// Mitsubishi GX Works2 project: plcgroup3_30_1   PLC: FX3G
// plcgroup3

// global labels: Global1
VAR_GLOBAL
  startDay AT X007 : BOOL;  (* מתחיל את היום *)
  ongoingDay AT Y007 : BOOL;  (* נורה שמציינת יום בתהליך *)
  endDay AT X011 : BOOL;  (* מתג סיום יום *)
  hold AT Y007 : BOOL;  (* ממסר החזקה לנורה Y7 *)
  analog_check AT X001 : BOOL;  (* מתג התחלת תהליך בישול *)
  lager AT M2 : BOOL;  (* ערך בינארי שמציין האם נבחר לייצר לאגר *)
  pilzner AT M3 : BOOL;  (* ערך בינארי שמציין האם נבחר לייצר פילסנר *)
  possible_manufacture_lager AT M4 : BOOL;  (* יהיה אחד אם ניתן לייצר לאגר מבחינת מלאי *)
  possible_manufacture_pilzner AT M5 : BOOL;  (* יהיה אחד אם ניתן לייצר פילסנר מבחינת מלאי *)
  cooking_In_process AT Y001 : BOOL;  (* נורה שמציינת שתהליך הבישול מתקיים *)
END_VAR
VAR_GLOBAL CONSTANT
  shmarim_Input_Amount : INT := 1000;  (* קבוע מלאי שמרים שיוזן בתחילת יום *)
  letet_Input_Amount : INT := 400;  (* קבוע מלאי לתת שיוזן בתחילת יום *)
  kashot_input_Amount : INT := 400;  (* קבוע מלאי קשות שיוזן בתחילת יום *)
END_VAR
VAR_GLOBAL
  shmarim_Inventory AT D1130 : INT;  (* רגיסטר שמחזיק בערך מלאי השמרים *)
  letet_Inventory AT D1140 : INT;  (* רגיסטר שמחזיק בערך מלאי הלתת *)
  kashot_Inventory AT D1150 : INT;  (* רגיסטר שמחזיק בערך מלאי הקשות *)
  total_beer_packs AT D1160 : INT;  (* רגיסטר שמחזיק בסך השישיות שיוצרו *)
  analog_Output AT D8282 : INT;  (* אנאלוג אאוטפוט *)
  analog_Input AT D8280 : INT;  (* אנאלוג אינפוט *)
  botteling_1Bottle AT X000 : BOOL;  (* מתג שמבקבק בקבוק אחד *)
  start_Botteling AT X002 : BOOL;  (* מתג שמתחיל בקבוק *)
  finish_Bottleing AT M7 : BOOL;  (* ממסר המציין סיום בקבוק *)
  six_Pack_Ligth AT Y002 : BOOL;  (* נורה שתדלק בזמן הבקבוק *)
END_VAR
VAR_GLOBAL CONSTANT
  constant5 : INT := 5;  (* קבוע 5 *)
END_VAR
VAR_GLOBAL
  cook_TIMER AT TC1 : BOOL;  (* משתנה לזמן הבישול *)
END_VAR
VAR_GLOBAL CONSTANT
  constant_40 : INT := 40;  (* מספר קבוע *)
  constant6 : INT := 6;  (* מספר קבוע *)
  pilzner_letet_6_req : INT := 6;  (* כמות לתת נדרשת לשישיית פילזנר *)
  pilzner_shmarim_6_req : INT := 120;  (* כמות שמרים נדרשת לשישיית פילזנר *)
  pilzner_kshot_6_req : INT := 54;  (* כמות קשות נדרשת לשישיית פילזנר *)
  lager_shmarim_6_req : INT := 150;  (* כמות שמרים נדרשת לשישיית לאגר *)
  lager_letet_6_req : INT := 12;  (* כמות לתת נדרשת לשישיית לאגר *)
  lager_kshot_6_req : INT := 60;  (* כמות קשות נדרשת לשישיית לאגר *)
END_VAR
VAR_GLOBAL
  finish_cooking_timer AT TS1 : BOOL;  (* מציין סיום בישול *)
  stast_tsisa AT X005 : BOOL;  (* מתג הפעלת תסיסה *)
  hivhov_round AT M8 : BOOL;  (* ממסר שיתחיל סבב הבהוב נוסף *)
  bulb3_on AT TC2 : BOOL;  (* הפעלת נורה 3 לצורך הבהוב *)
END_VAR
VAR_GLOBAL CONSTANT
  hivhov_time : INT := 5;  (* זמן הבהוב *)
END_VAR
VAR_GLOBAL
  bulb3_off AT TS2 : BOOL;  (* סיום טיימר נורה 3 בהבהוב *)
  bulb_y3 AT Y003 : BOOL;  (* נורה 3 *)
  bulb4_on AT TC3 : BOOL;  (* הפעלת נורה 4 לצורך הבהוב *)
  bulb4_off AT TS3 : BOOL;  (* סיום טיימר נורה 4 בהבהוב *)
  bulb_y4 AT Y004 : BOOL;  (* נורה 4 *)
  lager_tsisa_timer AT TC4 : BOOL;  (* טיימר לתסיסת הלאגר *)
END_VAR
VAR_GLOBAL CONSTANT
  lager_tsisa_time_3sec : INT := 30;  (* מספר קקבוע *)
  pilzner_tsisa_time_4sec : INT := 40;  (* מספר קבוע *)
END_VAR
VAR_GLOBAL
  pilzner_tsisa_timer AT TC5 : BOOL;  (* טיימר לתסיסת הפילסנר *)
  finish_tsisa_lager AT TS4 : BOOL;  (* סיום תסיסת הלאגר *)
  finish_tsisa_pilzner AT TS5 : BOOL;  (* סיום תסיסת הפילסנר *)
  start_cooking AT X001 : BOOL;  (* מתג התחלת בישול *)
  six_beers_packed AT CC1 : BOOL;  (* הבירות שנארזו בשישיה *)
END_VAR
VAR_GLOBAL CONSTANT
  constant_1 : INT := 1;  (* מספר קבוע *)
  constant_6 : INT := 6;
END_VAR
VAR_GLOBAL
  six_beers_packed_mimsar AT CS1 : BOOL;  (* סיום אריזת שישיה *)
  current_six_pack_packed AT CN1 : INT;  (* כמות הבירות הנוכחי שנארז בשישיה *)
  helper_for_first_itaration AT M9 : BOOL;  (* משתנה עזר שמציין איטרציה ראשונה *)
  mimsar_4_output AT M10 : BOOL;  (* ממסר להצגת אאוטפוט *)
END_VAR
VAR_GLOBAL CONSTANT
  contstant_10 : INT := 10;  (* מספר קבוע *)
END_VAR
VAR_GLOBAL
  end_iteration AT M17 : BOOL;  (* משתנה עזר לסיום איטרציה *)
  got_shmarim AT M20 : BOOL;  (* בודק אם יש שמרים לייצור לאגר *)
  got_letet AT M21 : BOOL;  (* בודק אם יש לתת לייצור לאגר *)
  got_kashot AT M22 : BOOL;  (* בודק אם יש קשות לייצור לאגר *)
  got_shmarim_p AT M30 : BOOL;  (* בודק אם יש שמרים לייצור פילסנר *)
  got_letet_p AT M31 : BOOL;  (* בודק אם יש לתת לייצור פילסנר *)
  got_kashot_p AT M32 : BOOL;  (* בודק אם יש קשות לייצור פילסנר *)
END_VAR
VAR_GLOBAL CONSTANT
  constant_5 : INT := 5;  (* מספר קבוע *)
END_VAR
VAR_GLOBAL
  analog_input_div400 AT D170 : INT;  (* רגיסטר שמעביר יחידות לאנאלוג אאוטפוט *)
  end_day_mimsar AT M40 : BOOL;  (* ממסר לסיום יום *)
  numOfOptionalLager AT D1170 : INT;  (* מספר אופטימלי לייצור של לאגר *)
  numOfOptionalPilzner AT D1180 : INT;  (* מספר אופטימלי לייצור של פילסנר *)
  theBestHarel AT M23 : BOOL;  (* הראל הגבר *)
END_VAR
VAR_GLOBAL CONSTANT
  constant4000 : INT := 4000;  (* מספר קבוע *)
  const400 : INT := 400;  (* מספר קבוע *)
  const0 : INT;  (* מספר קבוע *)
END_VAR

// task Task_01 (event TRUE, interval 0, priority 31): POU_01

PROGRAM POU_01
VAR
  update_shmarim_amount_lager : BOOL;
  update_amount_lager : BOOL;
END_VAR
(* structured ladder/FBD written out as ST: instructions are called as NAME(EN, inputs, outputs); _pN, _eN, _tN stand for wires *)
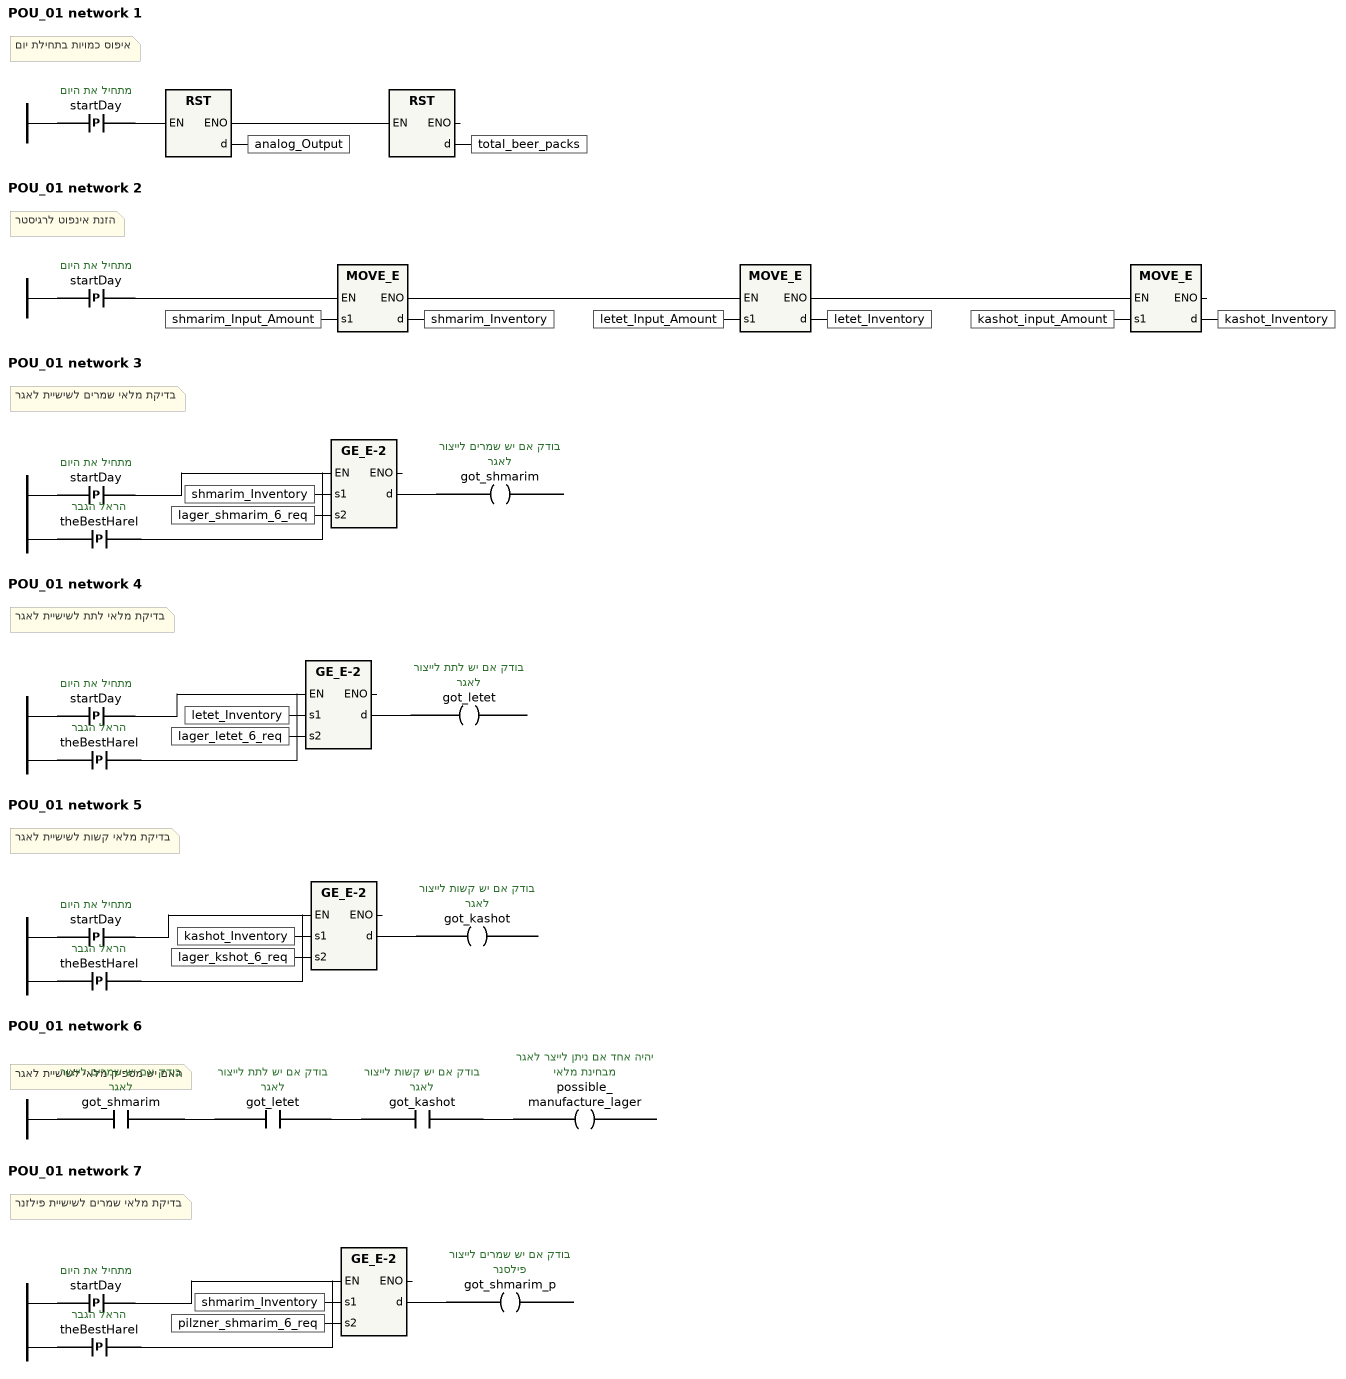
(* network 1 *)
(* איפוס כמויות בתחילת יום *)
_e1 := RST(LDP(TRUE, startDay), analog_Output);
RST(_e1, total_beer_packs);
(* network 2 *)
(* הזנת אינפוט לרגיסטר *)
_e1 := MOVE_E(LDP(TRUE, startDay), shmarim_Input_Amount, shmarim_Inventory);
_e2 := MOVE_E(_e1, letet_Input_Amount, letet_Inventory);
MOVE_E(_e2, kashot_input_Amount, kashot_Inventory);
(* network 3 *)
(* בדיקת מלאי שמרים לשישיית לאגר *)
GE_E(LDP(TRUE, startDay) OR LDP(TRUE, theBestHarel), shmarim_Inventory, lager_shmarim_6_req, _t1);
got_shmarim := _t1;
(* network 4 *)
(* בדיקת מלאי לתת לשישיית לאגר *)
GE_E(LDP(TRUE, startDay) OR LDP(TRUE, theBestHarel), letet_Inventory, lager_letet_6_req, _t1);
got_letet := _t1;
(* network 5 *)
(* בדיקת מלאי קשות לשישיית לאגר *)
GE_E(LDP(TRUE, startDay) OR LDP(TRUE, theBestHarel), kashot_Inventory, lager_kshot_6_req, _t1);
got_kashot := _t1;
(* network 6 *)
(* האם יש מספיק מלאי לשישיית לאגר *)
possible_manufacture_lager := got_shmarim AND got_letet AND got_kashot;
(* network 7 *)
(* בדיקת מלאי שמרים לשישיית פילזנר *)
GE_E(LDP(TRUE, startDay) OR LDP(TRUE, theBestHarel), shmarim_Inventory, pilzner_shmarim_6_req, _t1);
got_shmarim_p := _t1;
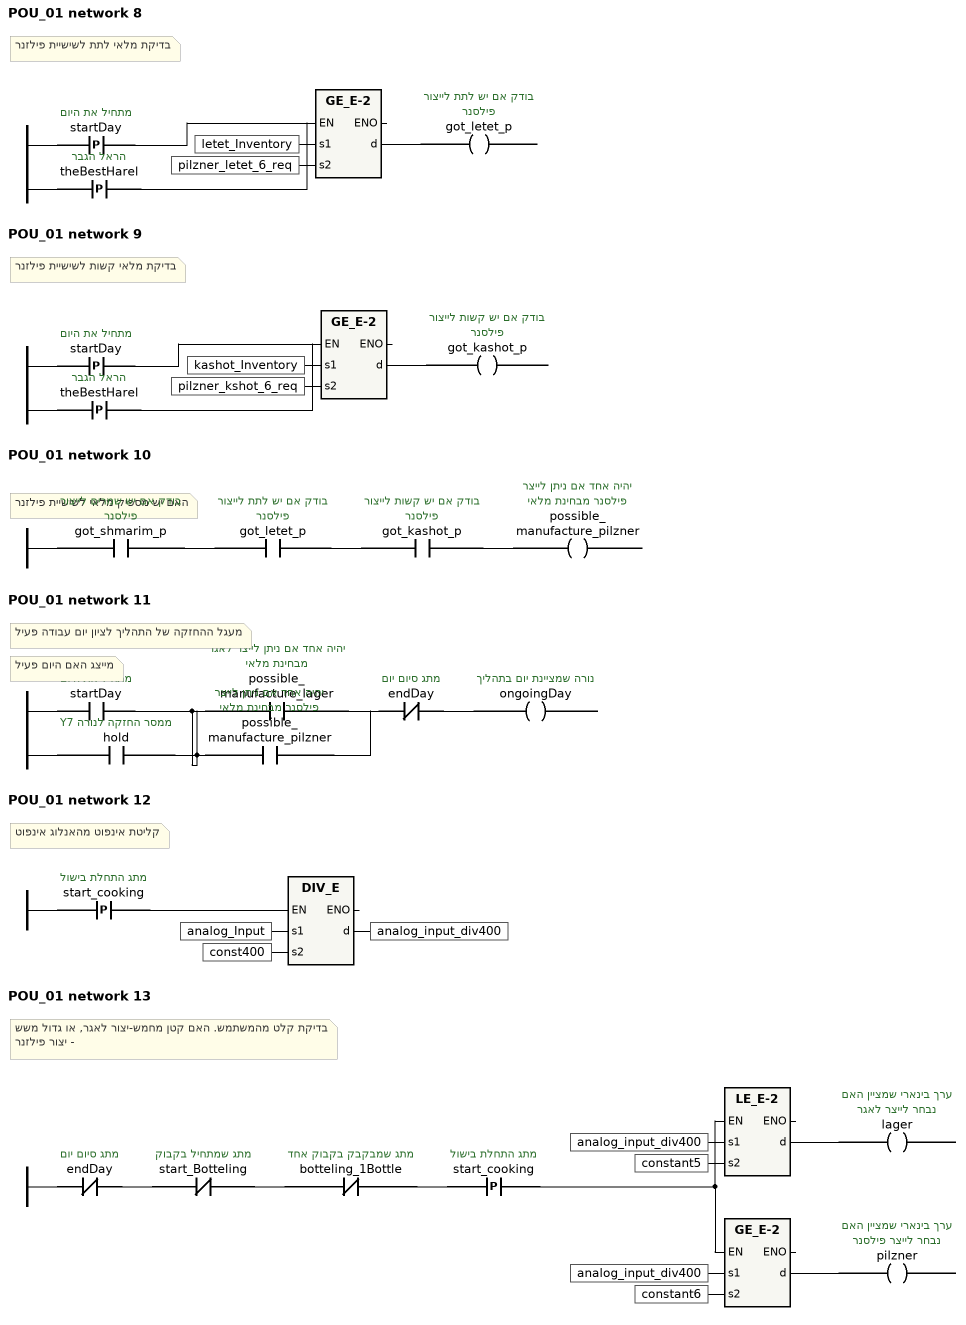
(* network 8 *)
(* בדיקת מלאי לתת לשישיית פילזנר *)
GE_E(LDP(TRUE, startDay) OR LDP(TRUE, theBestHarel), letet_Inventory, pilzner_letet_6_req, _t1);
got_letet_p := _t1;
(* network 9 *)
(* בדיקת מלאי קשות לשישיית פילזנר *)
GE_E(LDP(TRUE, startDay) OR LDP(TRUE, theBestHarel), kashot_Inventory, pilzner_kshot_6_req, _t1);
got_kashot_p := _t1;
(* network 10 *)
(* האם יש מספיק מלאי לשישיית פילזנר *)
possible_manufacture_pilzner := got_shmarim_p AND got_letet_p AND got_kashot_p;
(* network 11 *)
(* מעגל ההחזקה של התהליך לציון יום עבודה פעיל *)
(* מייצג האם היום פעיל *)
_p1 := startDay OR hold;
ongoingDay := ((_p1 AND possible_manufacture_lager) OR (_p1 AND possible_manufacture_pilzner)) AND NOT endDay;
(* network 12 *)
(* קליטת אינפוט מהאנלוג אינפוט *)
DIV_E(LDP(TRUE, start_cooking), analog_Input, const400, analog_input_div400);
(* network 13 *)
(* בדיקת קלט מהמשתמש. האם קטן מחמש-יצור לאגר, או גדול משש - יצור פילזנר *)
_p1 := NOT endDay AND NOT start_Botteling AND NOT botteling_1Bottle AND LDP(TRUE, start_cooking);
LE_E(_p1, analog_input_div400, constant5, _t2);
lager := _t2;
GE_E(_p1, analog_input_div400, constant6, _t3);
pilzner := _t3;
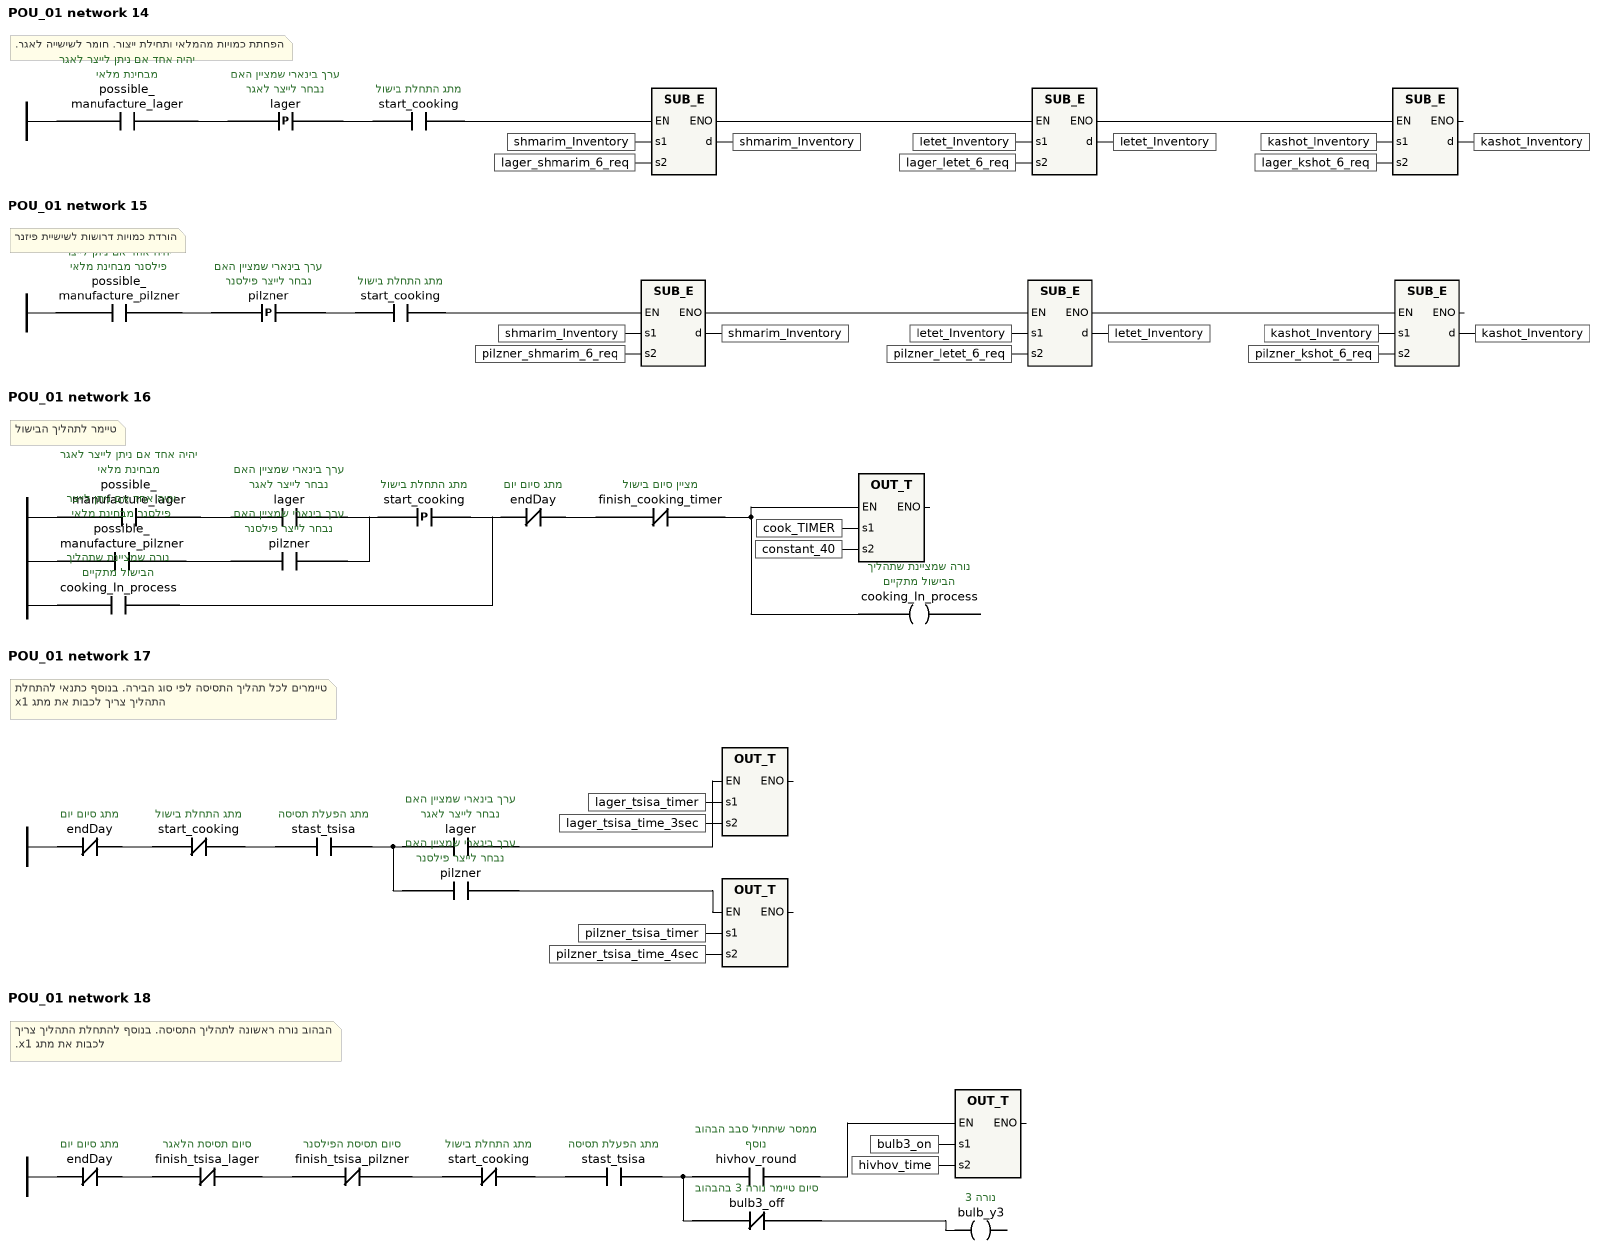
(* network 14 *)
(* הפחתת כמויות מהמלאי ותחילת ייצור. חומר לשישייה לאגר. *)
_e1 := SUB_E(possible_manufacture_lager AND LDP(TRUE, lager) AND start_cooking, shmarim_Inventory, lager_shmarim_6_req, shmarim_Inventory);
_e2 := SUB_E(_e1, letet_Inventory, lager_letet_6_req, letet_Inventory);
SUB_E(_e2, kashot_Inventory, lager_kshot_6_req, kashot_Inventory);
(* network 15 *)
(* הורדת כמויות דרושות לשישיית פיזנר *)
_e1 := SUB_E(possible_manufacture_pilzner AND LDP(TRUE, pilzner) AND start_cooking, shmarim_Inventory, pilzner_shmarim_6_req, shmarim_Inventory);
_e2 := SUB_E(_e1, letet_Inventory, pilzner_letet_6_req, letet_Inventory);
SUB_E(_e2, kashot_Inventory, pilzner_kshot_6_req, kashot_Inventory);
(* network 16 *)
(* טיימר לתהליך הבישול *)
_p1 := (((((possible_manufacture_lager AND lager) OR (possible_manufacture_pilzner AND pilzner)) AND LDP(TRUE, start_cooking)) OR cooking_In_process) AND NOT endDay) AND NOT finish_cooking_timer;
cooking_In_process := _p1;
OUT_T(_p1, cook_TIMER, constant_40);
(* network 17 *)
(* טיימרים לכל תהליך התסיסה לפי סוג הבירה. בנוסף כתנאי להתחלת התהליך צריך לכבות את מתג x1 *)
_p1 := NOT endDay AND NOT start_cooking AND stast_tsisa;
OUT_T(_p1 AND lager, lager_tsisa_timer, lager_tsisa_time_3sec);
OUT_T(_p1 AND pilzner, pilzner_tsisa_timer, pilzner_tsisa_time_4sec);
(* network 18 *)
(* הבהוב נורה ראשונה לתהליך התסיסה. בנוסף להתחלת התהליך צריך לכבות את מתג x1. *)
_p1 := NOT endDay AND NOT finish_tsisa_lager AND NOT finish_tsisa_pilzner AND NOT start_cooking AND stast_tsisa;
OUT_T(_p1 AND hivhov_round, bulb3_on, hivhov_time);
bulb_y3 := _p1 AND NOT bulb3_off;
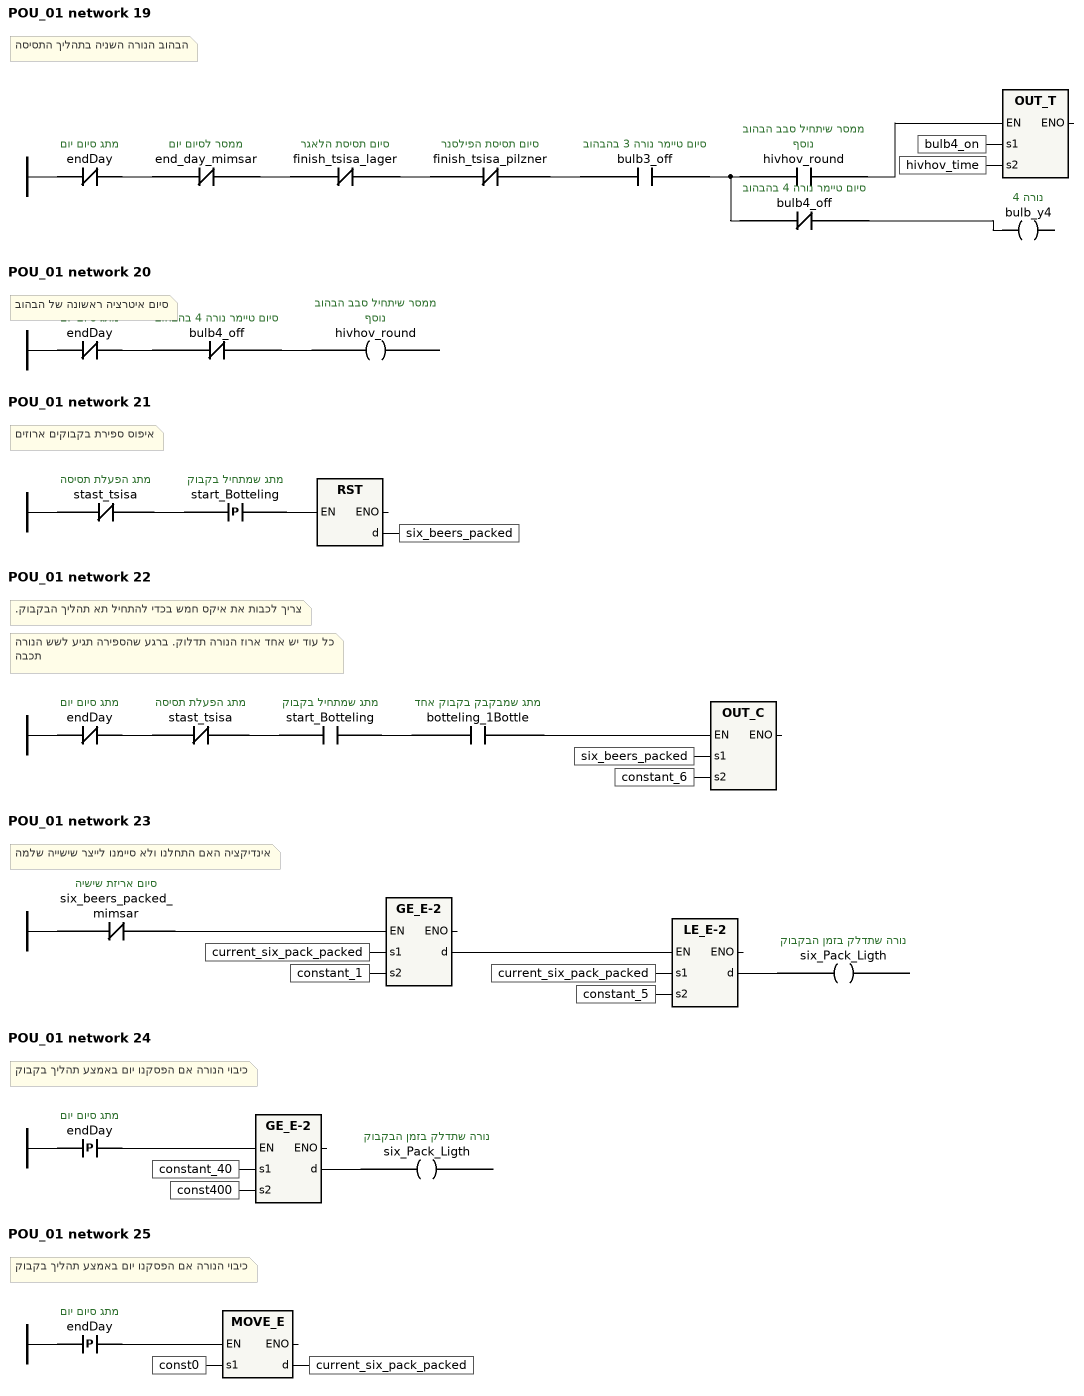
(* network 19 *)
(* הבהוב הנורה השניה בתהליך התסיסה *)
_p1 := NOT endDay AND NOT end_day_mimsar AND NOT finish_tsisa_lager AND NOT finish_tsisa_pilzner AND bulb3_off;
OUT_T(_p1 AND hivhov_round, bulb4_on, hivhov_time);
bulb_y4 := _p1 AND NOT bulb4_off;
(* network 20 *)
(* סיום איטרציה ראשונה של הבהוב *)
hivhov_round := NOT endDay AND NOT bulb4_off;
(* network 21 *)
(* איפוס ספירת בקבוקים ארוזים *)
RST(NOT stast_tsisa AND LDP(TRUE, start_Botteling), six_beers_packed);
(* network 22 *)
(* צריך לכבות את איקס חמש בכדי להתחיל תא תהליך הבקבוק. *)
(* כל עוד יש אחד ארוז הנורה תדלוק. ברגע שהספירה תגיע לשש הנורה תכבה *)
OUT_C(NOT endDay AND NOT stast_tsisa AND start_Botteling AND botteling_1Bottle, six_beers_packed, constant_6);
(* network 23 *)
(* אינדיקציה האם התחלנו ולא סיימנו לייצר שישייה שלמה *)
GE_E(NOT six_beers_packed_mimsar, current_six_pack_packed, constant_1, _t1);
LE_E(_t1, current_six_pack_packed, constant_5, _t2);
six_Pack_Ligth := _t2;
(* network 24 *)
(* כיבוי הנורה אם הפסקנו יום באמצע תהליך בקבוק *)
GE_E(LDP(TRUE, endDay), constant_40, const400, _t1);
six_Pack_Ligth := _t1;
(* network 25 *)
(* כיבוי הנורה אם הפסקנו יום באמצע תהליך בקבוק *)
MOVE_E(LDP(TRUE, endDay), const0, current_six_pack_packed);
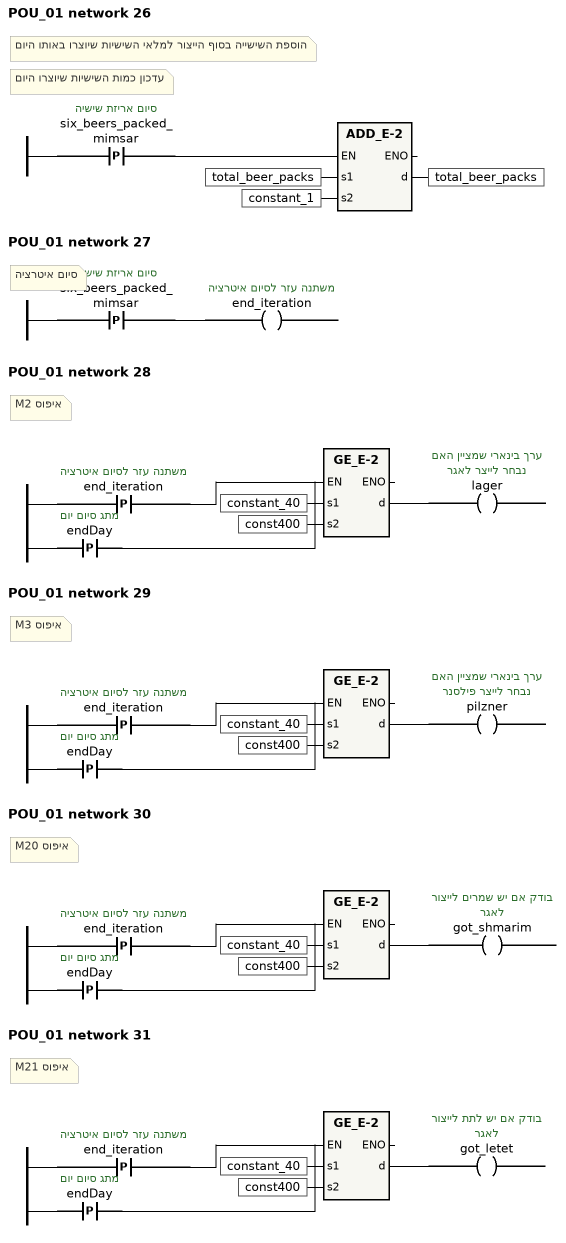
(* network 26 *)
(* הוספת השישייה בסוף הייצור למלאי השישיות שיוצרו באותו היום *)
(* עדכון כמות השישיות שיוצרו היום *)
ADD_E(LDP(TRUE, six_beers_packed_mimsar), total_beer_packs, constant_1, total_beer_packs);
(* network 27 *)
(* סיום איטרציה *)
end_iteration := LDP(TRUE, six_beers_packed_mimsar);
(* network 28 *)
(* איפוס M2 *)
GE_E(LDP(TRUE, end_iteration) OR LDP(TRUE, endDay), constant_40, const400, _t1);
lager := _t1;
(* network 29 *)
(* איפוס M3 *)
GE_E(LDP(TRUE, end_iteration) OR LDP(TRUE, endDay), constant_40, const400, _t1);
pilzner := _t1;
(* network 30 *)
(* איפוס M20 *)
GE_E(LDP(TRUE, end_iteration) OR LDP(TRUE, endDay), constant_40, const400, _t1);
got_shmarim := _t1;
(* network 31 *)
(* איפוס M21 *)
GE_E(LDP(TRUE, end_iteration) OR LDP(TRUE, endDay), constant_40, const400, _t1);
got_letet := _t1;
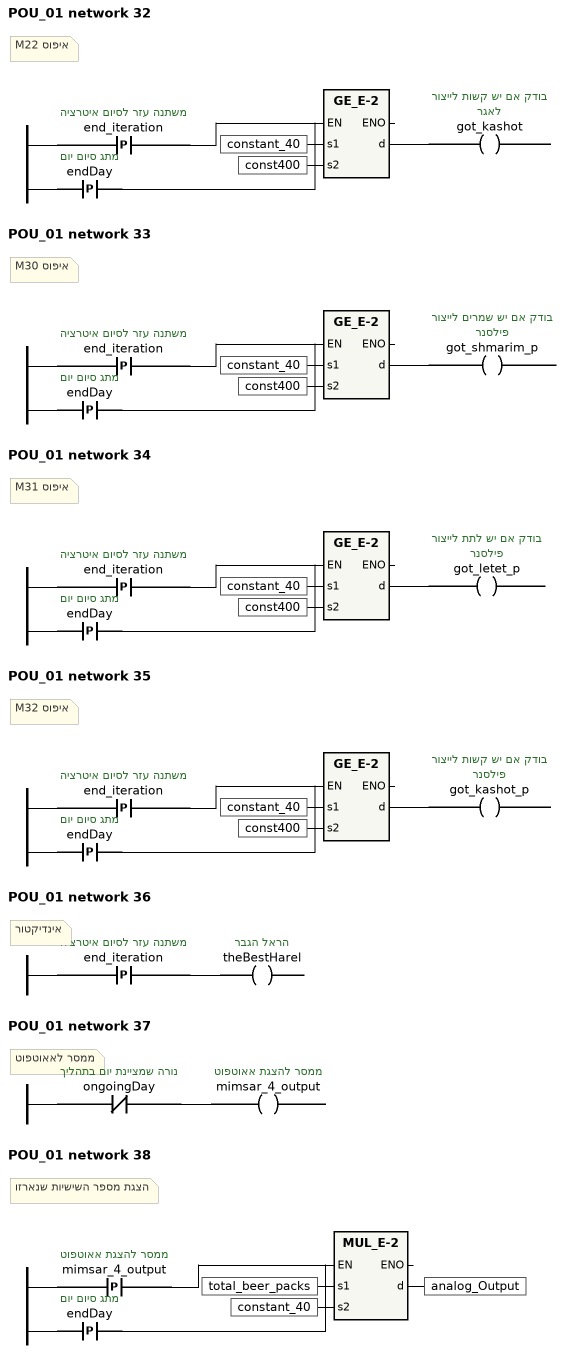
(* network 32 *)
(* איפוס M22 *)
GE_E(LDP(TRUE, end_iteration) OR LDP(TRUE, endDay), constant_40, const400, _t1);
got_kashot := _t1;
(* network 33 *)
(* איפוס M30 *)
GE_E(LDP(TRUE, end_iteration) OR LDP(TRUE, endDay), constant_40, const400, _t1);
got_shmarim_p := _t1;
(* network 34 *)
(* איפוס M31 *)
GE_E(LDP(TRUE, end_iteration) OR LDP(TRUE, endDay), constant_40, const400, _t1);
got_letet_p := _t1;
(* network 35 *)
(* איפוס M32 *)
GE_E(LDP(TRUE, end_iteration) OR LDP(TRUE, endDay), constant_40, const400, _t1);
got_kashot_p := _t1;
(* network 36 *)
(* אינדיקטור *)
theBestHarel := LDP(TRUE, end_iteration);
(* network 37 *)
(* ממסר לאאוטפוט *)
mimsar_4_output := NOT ongoingDay;
(* network 38 *)
(* הצגת מספר השישיות שנארזו *)
MUL_E(LDP(TRUE, mimsar_4_output) OR LDP(TRUE, endDay), total_beer_packs, constant_40, analog_Output);
END_PROGRAM
